// TIA Portal project "LAB1" (V16)

(* hardware
DEVICE "S71500/ET200MP station_2"  S7-1500 station
   slot 0: "Perfil soporte_0"  Rack  6ES7 590-1***0-0AA0
   slot 0: "PM 190W 120/230VAC"  PM 190W 120/230VAC  6EP1333-4BA00
   slot 1: "PLC_2"  CPU 1516-3 PN/DP  6ES7 516-3AN02-0AB0  V2.8
      slot 3: "Display de la CPU_1"  6ES7591-1BA00-0AA0
      slot 32768: "Interfaz PROFINET_1"  X1
         slot 32769: "Puerto_1"  X1 P1
         slot 32770: "Puerto_2"  X1 P2
      slot 33024: "Interfaz PROFINET_2"  X2
      slot 33280: "Interfaz DP_1"  X3
      slot 34817: "Virtual CP interface port_1"  Virtual CP interface port  Virtual CP interface port
   slot 2: "DI 32x24VDC HF_1"  DI 32x24VDC HF  6ES7 521-1BL00-0AB0  V2.0
   slot 3: "DQ 32x24VDC/0.5A HF_1"  DQ 32x24VDC/0.5A HF  6ES7 522-1BL01-0AB0  V1.0
   slot 4: "AI 8xU/I/RTD/TC ST_1"  AI 8xU/I/RTD/TC ST  6ES7 531-7KF00-0AB0  V2.0
   slot 5: "AQ 4xU/I ST_1"  AQ 4xU/I ST  6ES7 532-5HD00-0AB0  V2.0
*)

// ===== PLC "PLC_2"  CPU 1516-3 PN/DP =====

VAR_GLOBAL   // PLC tag table "Tabla de variables estándar"
   "A" AT %M0.0 : Bool;
   "B" AT %M0.1 : Bool;
   "AND" AT %Q0.0 : Bool;
   "OR" AT %Q0.1 : Bool;
   "XOR" AT %Q0.2 : Bool;
   "NOT" AT %Q0.3 : Bool;
END_VAR

FUNCTION "KOP" : Void   // FC1, LAD
{ S7_Optimized_Access := 'TRUE' }
VERSION : 0.1
// KOP
BEGIN

REGION Network 1
   // AND
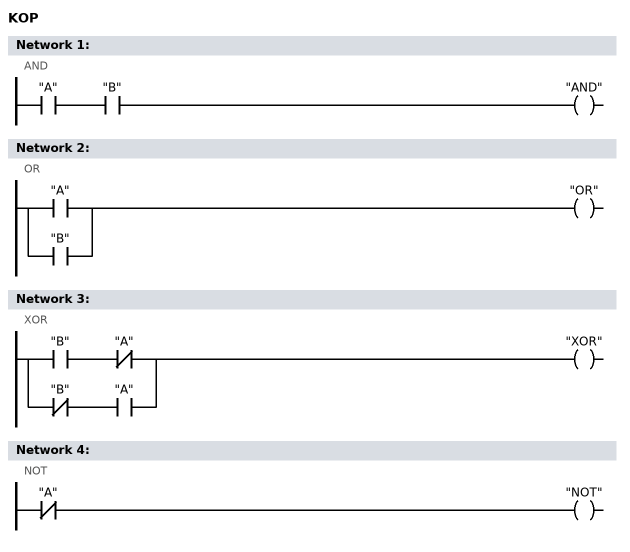
   RUNG wire#powerrail
      Contact( "A" )
      Contact( "B" )
      Coil( "AND" )
   END_RUNG
   // the same network as SCL:
   "AND" := "A" AND "B";
END_REGION

REGION Network 2
   // OR
   RUNG wire#powerrail
      Contact( "A" )
      wire#w1
      Coil( "OR" )
   END_RUNG
   RUNG wire#powerrail
      Contact( "B" )
   END_RUNG wire#w1
   // the same network as SCL:
   "OR" := "A" OR "B";
END_REGION

REGION Network 3
   // XOR
   RUNG wire#powerrail
      Contact( "B" )
      I_Contact( "A" )
      wire#w1
      Coil( "XOR" )
   END_RUNG
   RUNG wire#powerrail
      I_Contact( "B" )
      Contact( "A" )
   END_RUNG wire#w1
   // the same network as SCL:
   "XOR" := ("B" AND NOT "A") OR (NOT "B" AND "A");
END_REGION

REGION Network 4
   // NOT
   RUNG wire#powerrail
      I_Contact( "A" )
      Coil( "NOT" )
   END_RUNG
   // the same network as SCL:
   "NOT" := NOT "A";
END_REGION
END_FUNCTION

FUNCTION "FUP" : Void   // FC2, FBD
{ S7_Optimized_Access := 'TRUE' }
VERSION : 0.1
// FUP
BEGIN

REGION Network 1
   // AND
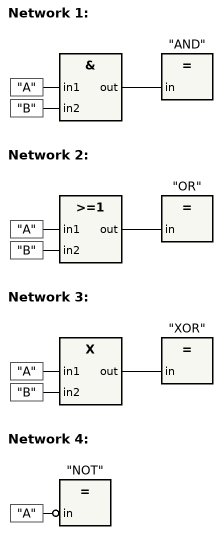
   "AND" := "A" AND "B";
END_REGION

REGION Network 2
   // OR
   "OR" := "A" OR "B";
END_REGION

REGION Network 3
   // XOR
   "XOR" := "A" XOR "B";
END_REGION

REGION Network 4
   // NOT
   "NOT" := NOT "A";
END_REGION
END_FUNCTION

FUNCTION "AWL" : Void   // FC3, STL
{ S7_Optimized_Access := 'TRUE' }
VERSION : 0.1
// AWL
BEGIN

REGION Network 1
   // AND
         A     "A";
         A     "B";
         =     "AND";
END_REGION

REGION Network 2
   // OR
         O     "A";
         O     "B";
         =     "OR";
END_REGION

REGION Network 3
   // XOR
         X     "A";
         X     "B";
         =     "XOR";
END_REGION

REGION Network 4
   // NOT
         ON    "A";
         =     "NOT";
END_REGION
END_FUNCTION

FUNCTION "SCL" : Void   // FC4, SCL
{ S7_Optimized_Access := 'TRUE' }
VERSION : 0.1
BEGIN
   "AND" := "A" AND "B";
   "OR" := "A" OR "B";
   "XOR" := "A" XOR "B";

   IF "A" = TRUE THEN
       "NOT" := FALSE;
   ELSE
       "NOT" := TRUE;
   END_IF;
END_FUNCTION

ORGANIZATION_BLOCK "Main"   // OB1, LAD, ProgramCycle
TITLE = "Main Program Sweep (Cycle)"
{ S7_Optimized_Access := 'TRUE' }
VERSION : 0.1
   VAR_INPUT
      Initial_Call : Bool;   // Initial call of this OB
      Remanence : Bool;   // =True, if remanent data are available
   END_VAR
BEGIN

REGION Network 1
   // KOP
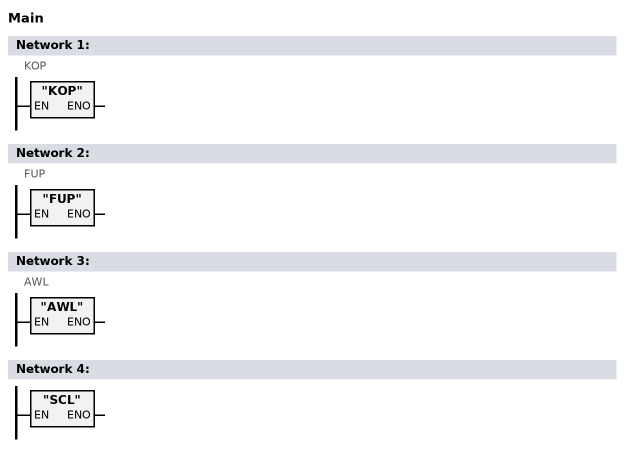
   RUNG wire#powerrail
      "KOP"()
   END_RUNG
   // the same network as SCL:
   "KOP"();
END_REGION

REGION Network 2
   // FUP
   RUNG wire#powerrail
      "FUP"()
   END_RUNG
   // the same network as SCL:
   "FUP"();
END_REGION

REGION Network 3
   // AWL
   RUNG wire#powerrail
      "AWL"()
   END_RUNG
   // the same network as SCL:
   "AWL"();
END_REGION

REGION Network 4
   RUNG wire#powerrail
      "SCL"()
   END_RUNG
   // the same network as SCL:
   "SCL"();
END_REGION
END_ORGANIZATION_BLOCK